FUNCTION_BLOCK FB_Maschinentuer
VAR_INPUT
	//Sensor Eingang
	bDoorC : BOOL;
	bDoorO : BOOL;
	//Steuereingänge
	bEnable : Bool; //Freigabe für Maschinentür
	bOpen : BOOL;
	bClose : BOOL;
END_VAR
VAR_OUTPUT
	//Aktor Ausgang
	bVentil : BOOL;
	//Zustädne
	bError : BOOL;
END_VAR
VAR
	nState: INT := 0;
END_VAR

Case nstate OF
	0: // Tür geschlossen
	// Ausgänge
	bVentil := TRUE;
	
	//Übergangsbedingung
	IF NOT bDoorC AND bEnable THEN
		nState := 3; //Tür schließen
	ELSIF bOpen THEN
		nState := 1; // Tür öffnen 
	END_IF
	
	1: // Tür öffnen
	//Ausgänge setzten
	bVentil := FALSE;
	
	//Übergangsbedingung
	IF bDoorO THEN
		nState := nState + 1; //Tür geöffnet
	END_IF
	
	2: // Tür geöffnet
	bVentil := FALSE;
	
	IF bClose AND bEnable THEN
		nState := 3; // Tür schließen
	END_IF
	
	3: //Tür schließen
	bVentil := TRUE;
	IF bDoorC THEN
		nState := 0;
	END_IF
END_CASE

END_FUNCTION_BLOCK

(* stored: Version 1.1.0.1, ProductVersion 3.1.4024.15
   POU FB_Maschinentuer: Id {2fb64f53-bf99-4ab3-8476-84085422f959}, SpecialFunc None *)
